PROGRAM MAIN
VAR
    _tcoTestContext : TcoTestContext;
    _wpfContext : WpfContext;
    _wpfContextCall : BOOL := FALSE;
END_VAR

_tcoTestContext.ProbeRun();

IF _wpfContextCall THEN
    _wpfContext.Run();
END_IF

END_PROGRAM

(* stored: Version 1.1.0.1, ProductVersion 3.1.4024.12
   POU MAIN: Id {04a19911-77de-0523-3700-ac8476e9a3fc}, SpecialFunc None *)
